{attribute 'linkalways'} 
{attribute 'no_explicit_call' := 'This FB is a CLASS and must be accessed using methods or properties'}
{attribute 'enable_dynamic_creation'}
FUNCTION_BLOCK WriteBitToBoolOperation EXTENDS Disposable IMPLEMENTS I_DatatypeOperation
VAR
	source : I_BIT;
	destination : REFERENCE TO _BOOL;
END_VAR

METHOD Execute
VAR
END_VAR
destination.Value := source.Value;
END_METHOD

METHOD FB_init : BOOL
VAR_INPUT
	bInitRetains : BOOL; // if TRUE, the retain variables are initialized (warm start / cold start)
	bInCopyCode : BOOL;  // if TRUE, the instance afterwards gets moved into the copy code (online change)
	Source : I_BIT;
	Destination : REFERENCE TO _BOOL;
END_VAR
THIS^.source := Source;
THIS^.destination REF= Destination;
END_METHOD

END_FUNCTION_BLOCK

(* stored: Version 1.1.0.1, ProductVersion 3.1.4024.15
   POU WriteBitToBoolOperation: Id {f79428c6-f25e-4318-941a-ed0037d31ddf}, SpecialFunc None
   Folder Constructor: Id {777f1816-6c52-43ff-9b5b-bb4f767dc76a}
   Method Execute: Id {0ea8cbde-5d5d-4d0e-babc-0a1efe9db281}
   Method FB_init: Id {5d6dabf3-8c3a-49c4-8c4e-7da29ad475f3} *)
